// TIA Portal V19 export
TYPE "Prod_Item"
// stored: Access Published
   STRUCT
      O_ID : DInt;   // ID PLC per riferimento allìordine di produzione
      "Type" : Int;   // 1= Caricato da MES; 2= Caricamento HMI manuale
      Status : Int;   // 0 = Non iniziato; 1 = Iniziato; 2 = In lavoro; 3 = Conclusione Parziale; 4 = Concluso completo; 5 = Concluso complerto; 6 = Pausa parziale; 7 = Pausa totale
      Status_Saved : Int;   // Stato salvato = Su variazione rispetto a "Status" sono inviati messaggi a MES
      Material_Len_REQ : Real;   // Quanto materiale è richiesto per eseguire l'ordine
      Material_Len_ToGo : Real;   // Quanto materiale manca per concludere l'ordine
      MES_IDP : String[30];   // ID MES per riferimento all'ordine di prosuzione
      MES_Profile_Code : String[3];   // Codice profilo dei pezzi da produrre: profilo accoppiato a C (sigla codice S); profilo semiguscio SG (sigla codice G)
      MES_PPrf_Name : String[20];   // Nome dell programma profilo richiesto da MES (es.C040x45x1.25)
      PPrf_No : DInt;   // Numero del programma profillo che corrisponde al codice MES del prodotto da eseguire
      Beam_Code : Int;   // Codice Pezzo: 0= SG formato da una singola parte; 1= C/S = Formato da due parti accoppiate
      Beams_W_A : Real;   // Dim. base pezzo (W) = Altezza in impilamento (A)
      Beams_H_B : Real;   // Dim. altezza pezzo (H) = base in impilamento (B)
      Beams_Thickness : Real;   // Spessore lamiera del profilo
      Beams_Len_Min : Real;   // Lunghezza pezzo - Tolleranza minima
      Beams_Len_Max : Real;   // Lunghezza pezzo + Tolleranza massima
      Beams_Len : Real;   // Lunghezza pezzi richiesta
      Beams_REQ : DInt;   // Quantità di pezzi da produrre
      Beams_ToGo : DInt;   // Quante pezzi mancano per concludere l'ordine
      Beams_NonConforming : DInt;   // Somma Beams_NG + Beams_TOCHECK
      Beams_GOOD : DInt;   // Pezzi prodotti con qualità CONFORMI (2 parti = 1 pezzo)
      Beams_GOOD_R : DInt;   // Pezzi prodotti con qualità CONFORMI dopo il RICONIDZIONAMENTO
      Beams_NG : DInt;   // Pezzi prodotti con qualità NG = Scartati dopo controllo qualità
      Beams_TOCHECK : DInt;   // Pezzi prodotti che attendono controllo qualità
      Parts_Len : Real;   // Lunghezza delle parti con target al centro della tolleranza richiesta
      Parts_Tol : Real;   // Tolleranza su lunghezza parte tagliata
      Parts_REQ : DInt;   // Quantità di parti da produrre (2 parti = 1 pezzo)
      Parts_ToGo : DInt;   // Quante parti mancano per concludere l'ordine
      Parts_NonConforming : DInt;   // Somma Parts_NG + Parts_TOCHECK
      Parts_GOOD : DInt;   // Parti prodotte con qualità CONFORMI (parte = semilavorato = guscio)
      Parts_GOOD_R : DInt;   // Parti prodotte con qualità CONFORMI dopo il ricondizinamento
      Parts_NG : DInt;   // Parti prodotte con qualità NG = Scartati dopo controllo qualità + eseguiti scarte
      Parts_TOCHECK : DInt;   // Parti prodotte che attendono controllo qualità
      Kanban_Style : Bool;   // Ordine tipo kanban = senza limitazione dul numero di pezzi da produrre
      Use_Ribbing_Roll : Bool;   // Eseguire nervatura su profilo
      Use_Trace_Mark_Tool : Bool;   // I pezzi devano avere il marchio di tracciabilità (Lotto / Colata)
      Use_Thick_Mark_Tool : Bool;   // I pezzi devono avere il marchio MODULBLOK con identificazione dello spessore lamiera
      PackLayout_BeamsPerLayer : Int;   // Schema del pacco - Numero pezzi per strato
      PackLayout_Layers_Qty : Int;   // Schema del pacco - Numero strati
   END_STRUCT;
END_TYPE
